(* PLC project Generated.project, CODESYS CODESYS V3.5 SP19 Patch 1 *)
(* stored: creationDateTime 2026-09-14T14:47:22.359825, modificationDateTime 2026-09-14T14:47:22.359825 *)

(* values of E_CycleDepthStopMode: KOBOLD_ONLY: Comportement historique : fond valide par DI Kobold; SETPOINT_ONLY: Arret sur consigne de profondeur valide; KOBOLD_OR_SETPOINT: Premier evenement valide des deux *)

{attribute 'qualified_only'}
{attribute 'strict'}
TYPE E_CycleDepthStopMode : (KOBOLD_ONLY := 0, SETPOINT_ONLY := 1, KOBOLD_OR_SETPOINT := 2);
END_TYPE
